(* PLC project motors, Dassault Systèmes ControlBuild 2024x *)
(* stored: creationDateTime 2023-10-03T11:13:47-01:00 *)

FUNCTION_BLOCK tni_clock.motors
  VAR_INPUT
    stepMotorSecond : BOOL := false;
    stepMotorMinute : BOOL := false;
    stepMotorHour : BOOL := false;
  END_VAR
  VAR
    hourHand : INT := 0;
    minuteHand : INT := 0;
    secondHand : INT := 0;
  END_VAR

(** Calculation of degrees hands positions for the animation**)


IF RE stepMotorHour THEN
	hourHand := hourHand + 360/12;
	IF hourHand >= 360 THEN hourHand:=0; END_IF;
END_IF;
IF RE stepMotorMinute THEN
	minuteHand:= minuteHand+ 360/60;
	IF minuteHand >= 360 THEN minuteHand:=0; END_IF;
END_IF;
IF RE stepMotorSecond THEN
	secondHand:= secondHand + 360/60;
	IF secondHand >= 360 THEN secondHand:=0; END_IF;
END_IF;
END_FUNCTION_BLOCK
